SUBAPPLICATION Uebung_007d2 (* Blinker mit E_CYCLE und E_T_FF *)
  (* Standard: 61499-2; Description: Copyright (c) 2023 Meisterschulen am Ostbahnhof This program and the accompanying materials are made available under the terms of the Eclipse Public License 2.0 which is available at https://www.eclipse.org/legal/epl-2.0/ SPDX-License-Identifier: EPL-2.0 *)
  (* Version 1.0, 2023-10-23, Franz Höpfinger, Meisterschulen am Ostbahnhof, initial API and implementation and/or initial documentation *)
  PACKAGE Uebungen;
  IMPORT logiBUS::io::DQ::logiBUS_DO::Output_Q1;
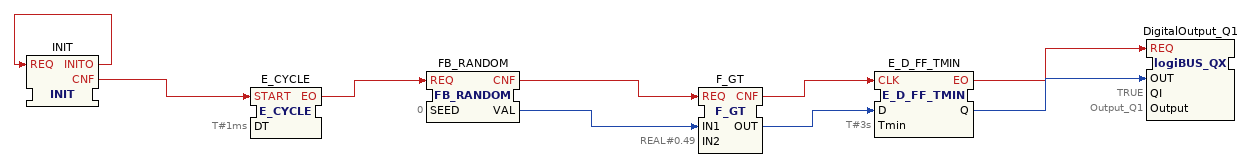
  FBS
    DigitalOutput_Q1 : logiBUS::io::DQ::logiBUS_QX(QI := TRUE, Output := Output_Q1);
    E_CYCLE : iec61499::events::E_CYCLE(DT := T#1ms);
    FB_RANDOM : eclipse4diac::utils::FB_RANDOM(SEED := 0);
    F_GT : iec61131::comparison::F_GT(IN2 := REAL#0.49);
    E_D_FF_TMIN : iec61499::events::E_D_FF_TMIN(Tmin := T#3s);
    INIT : iec61131::booleanOperators::INIT;
  END_FBS
  EVENT_CONNECTIONS
    E_CYCLE.EO TO FB_RANDOM.REQ;
    FB_RANDOM.CNF TO F_GT.REQ;
    F_GT.CNF TO E_D_FF_TMIN.CLK;
    E_D_FF_TMIN.EO TO DigitalOutput_Q1.REQ;
    INIT.INITO TO INIT.REQ;
    INIT.CNF TO E_CYCLE.START;
  END_CONNECTIONS
  DATA_CONNECTIONS
    FB_RANDOM.VAL TO F_GT.IN1;
    F_GT.OUT TO E_D_FF_TMIN.D;
    E_D_FF_TMIN.Q TO DigitalOutput_Q1.OUT;
  END_CONNECTIONS
END_SUBAPPLICATION
